// TIA Portal V21 export
TYPE "OBJ_Fw_Error_V200_Type"
   STRUCT
      f32_KP_FollowError { ExternalVisible := 'False'} : Real;
      f32_LastPosition { ExternalVisible := 'False'} : Real;
      f32_LastFollowError { ExternalVisible := 'False'} : Real;
   END_STRUCT;
END_TYPE
